// TIA Portal V16 export
// export: Created 2021-11-12T13:32:53.7755937Z, ExportSetting WithDefaults, DisplayName Totally Integrated Automation Portal, DisplayVersion V16 Update 3, DisplayName TIA Portal Version Control Interface, DisplayVersion V16 Update 2, DisplayName TIA Portal Openness, DisplayVersion V16 Update 3, DisplayName SINAMICS Startdrive Advanced, DisplayVersion V16 Update 5, DisplayName SINAMICS Startdrive G130, G150, S120, S150, SINAMICS MV, S210, DisplayVersion V16 Update 5, DisplayName SINAMICS Startdrive G110M, G120, G120C, G120D, G120P, G115D, DisplayVersion V16 Update 5, DisplayName STEP 7 Professional, DisplayVersion V16 Update 3, DisplayName STEP 7 Safety, DisplayVersion V16, DisplayName WinCC UA Professional, DisplayVersion V16 Update 3
DATA_BLOCK "HMI_CMD_BSN4"   // DB71
{ S7_Optimized_Access := 'TRUE' }
VERSION : 0.1
// stored: AutoNumber true, DBAccessibleFromOPCUA true, IsOnlyStoredInLoadMemory false, IsRetainMemResEnabled false, IsWriteProtectedInAS false, MemoryReserve 100
   VAR
      xxxxx___BinarySensors___xxxxx : Byte;
      xxxxx___BinaryOthers___xxxxx : Byte;
      xxxxx___AnalogueSensors___xxxxx : Byte;
      xxxxx___Drives___xxxxx : Byte;
      xxxxx___Others___xxxxx : Byte;
      Commands : "UDT_BSN_Command";   // Material flow commands
      xxxxx___SensorAlarms___xxxxx : Byte;
      Furnace_Alarm : "UDT_DI_Mon_Command";   // from furnace
      LiveBit_Alarm : "UDT_DI_Mon_Command";   // communication
      DataTracking_Alarm : "UDT_DI_Mon_Command";   // part on senzor is not in data tracking
      Senzor_Alarm : "UDT_DI_Mon_Command";   // part in data tracking is not on senzor
      Alarm_5 : "UDT_DI_Mon_Command";
      Alarm_6 : "UDT_DI_Mon_Command";
      Alarm_7 : "UDT_DI_Mon_Command";
      Alarm_8 : "UDT_DI_Mon_Command";
      ES { S7_SetPoint := 'True'} : "UDT_DI_Mon_Command";   // E-stop BSN4 and BSN5
      xxxxx___ProcessAlarms___xxxxx : Byte;
   END_VAR
BEGIN
END_DATA_BLOCK
